INTERFACE I_Timestamp

METHOD PUBLIC IsDurationElapsed : BOOL
VAR_INPUT
	Duration : TIME;
END_VAR
END_METHOD

PROPERTY PUBLIC TimeSince : TIME
GET
END_GET
END_PROPERTY

END_INTERFACE

(* stored: Version 1.1.0.1, ProductVersion 3.1.4024.12
   Itf I_Timestamp: Id {cda42b70-ee0a-01ec-339c-c264e0149db9}
   Method IsDurationElapsed: Id {ee250b15-aa7f-064a-29b9-5b21e87a7149}
   Property TimeSince: Id {798c4094-5997-0a6a-04ca-7eee52ed2a40}
   Get Get: Id {0df1e69a-e95d-0b42-2ff7-a939ec21dbe4} *)
